# EPICS substitutions: viocs/si_ps/si_psApp/Db/sda1.substitutions
file "db/individual.db" {
    pattern { family, pos, num }
        { "SDA1", "01C1", "" }
        { "SDA1", "04C4", "" }
        { "SDA1", "05C1", "" }
        { "SDA1", "08C4", "" }
        { "SDA1", "09C1", "" }
        { "SDA1", "12C4", "" }
        { "SDA1", "13C1", "" }
        { "SDA1", "16C4", "" }
        { "SDA1", "17C1", "" }
        { "SDA1", "20C4", "" }
}
